// TIA Portal V18 export
DATA_BLOCK "FB2-meteringpgmFB_DB"   // DB59
VERSION : 0.1
// stored: AutoNumber true, DBAccessibleFromOPCUA true, InstanceOfName FB2-meteringFB, InstanceOfType FB
"FB2-meteringFB"
   // VAR_INPUT
   //    Metering_function : Int;
   //    "DO Continuous metering" : Bool;
   //    Dispensing_time : DInt;
   //    "Set Qty in ml" : Real;
   //    "VC1 Pulses" : DInt;
   //    "VC2 Pulses" : DInt;
   //    VC1_impulse : Real;
   //    VC2_impulse : Real;
   //    "Outlet Open  to Pump ON A delay" : DInt;
   //    "Outlet Open  to Pump ON B delay" : DInt;
   //    "Pump Off  to Inlet A Close" : DInt;
   //    "Pump Off  to Inlet B Close" : DInt;
   //    "Mixer ON to Outlet ON" : DInt;
   //    "Pump Off  to Outlet Close" : DInt;
   //    "Outlet Close to Mixer Off" : DInt;
   // END_VAR
   // VAR_OUTPUT
   //    "Volume dispensed" : Real;
   //    "Run time" : Int;
   // END_VAR
   // VAR_IN_OUT
   //    ON_inlet_A : Bool;
   //    ON_inlet_B : Bool;
   //    ON_Pump_A : Bool;
   //    ON_pump_B : Bool;
   //    ON_valve_A : Bool;
   //    ON_valve_B : Bool;
   //    ON_Mixer : Bool;
   //    "Start Metering" : Bool;
   //    "Stop metering" : Bool;
   //    "Process running" : Bool;
   //    "process completed" : Bool;
   // END_VAR
   // VAR
   //    "pump A to valveA delay" : Bool;
   //    "Pump B to valve B delay" : Bool;
   //    "Pump Off to mixer off delay_1" : Bool;
   //    "VC1 pulses prev" : DInt;
   //    "VC2 pulses prev" : DInt;
   //    "VC1 pulse generted" : DInt;
   //    "VC2 pulse generated" : DInt;
   //    "Pump A Voulme dispensed" : Real;
   //    "Pump B volume dispensed" : Real;
   //    "Total Volume dispensed" : Real;
   //    "metering started" : Bool;
   //    "metering time in msec" : DInt;
   //    "dispense time elapsed" : Bool;
   //    R_TRIG_Instance { S7_SetPoint := 'True'} : R_TRIG;
   //    IEC_Timer_0_Instance { S7_SetPoint := 'True'} : TON_TIME;
   //    IEC_Timer_0_Instance_1 { S7_SetPoint := 'True'} : TON_TIME;
   //    IEC_Timer_0_Instance_2 { S7_SetPoint := 'True'} : TON_TIME;
   //    R_TRIG_Instance_1 { S7_SetPoint := 'True'} : R_TRIG;
   //    temp { S7_SetPoint := 'True'} : Bool;
   //    IEC_Timer_0_Instance_3 { S7_SetPoint := 'True'} : TON_TIME;
   //    IEC_Timer_0_Instance_4 { S7_SetPoint := 'True'} : TON_TIME;
   //    IEC_Timer_0_Instance_5 { S7_SetPoint := 'True'} : TON_TIME;
   //    IEC_Timer_0_Instance_6 { S7_SetPoint := 'True'} : TON_TIME;
   //    IEC_Timer_0_Instance_7 { S7_SetPoint := 'True'} : TON_TIME;
   //    IEC_Timer_0_Instance_8 { S7_SetPoint := 'True'} : TON_TIME;
   // END_VAR
BEGIN
END_DATA_BLOCK
